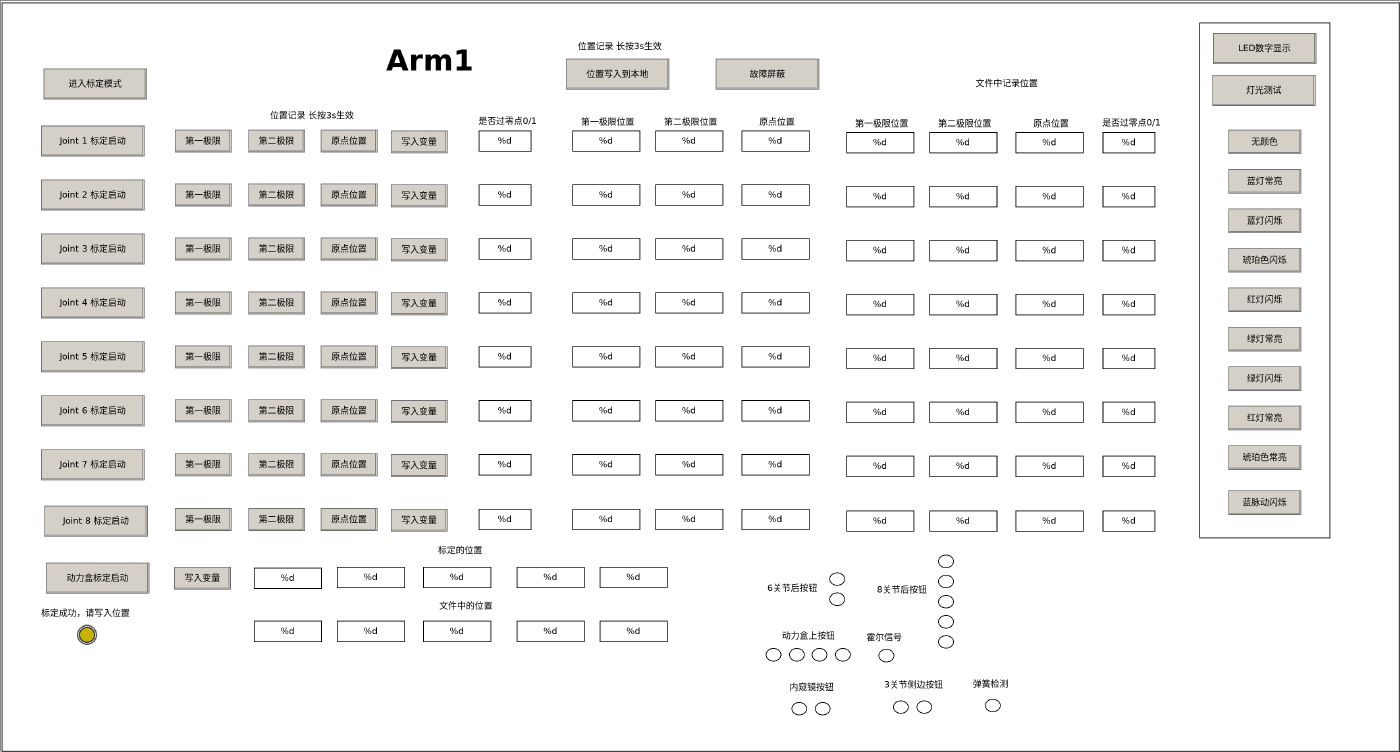
VISUALIZATION arm1Cail  // 1737x934
    Rectangle (2,3 1735x931)
    Button (54,85 128x38), "进入标定模式", colour toggle: GVL_armCali.g_armEnterCaliMode[1]
        toggle GVL_armCali.g_armEnterCaliMode[1]
    Button (51,156 128x38), "Joint 1 标定启动", colour toggle: GVL_armCali.g_jointIntoCaliState[1][1]
        toggle GVL_armCali.g_jointIntoCaliState[1][1]
    Label (435,49 197x52), "Arm1"
    Button (51,223 128x38), "Joint 2 标定启动", colour toggle: GVL_armCali.g_jointIntoCaliState[1][2]
        toggle GVL_armCali.g_jointIntoCaliState[1][2]
    Button (217,161 70x28), "第一极限", colour toggle: GVL_armCali.g_linkEncFristCaliTrigger[1][1]
        tap GVL_armCali.g_linkEncFristPosCali[1][1]
    Button (308,161 70x28), "第二极限", colour toggle: GVL_armCali.g_linkEncSecondCaliTrigger[1][1]
        tap GVL_armCali.g_linkEncSecondPosCali[1][1]
    Rectangle (594,162 65x26), "%d", text variable: GVL_armCali.g_linkZeroCrossOrNot[1][1]
    Label (589,139 82x23), "是否过零点0/1"
    Rectangle (710,162 84x26), "%d", text variable: GVL_armCali.g_linkLimitFristPos[1][1]
    Label (713,140 82x23), "第一极限位置"
    Rectangle (813,162 84x26), "%d", text variable: GVL_armCali.g_linkLimitSecondPos[1][1]
    Label (816,140 82x23), "第二极限位置"
    Label (312,132 150x23), "位置记录 长按3s生效"
    Rectangle (920,162 84x26), "%d", text variable: GVL_armCali.g_linkHomePos[1][1]
    Label (923,140 82x23), "原点位置"
    Button (398,161 70x28), "原点位置", colour toggle: GVL_armCali.g_linkEncHomePosCaliTrigger[1][1]
        tap GVL_armCali.g_linkEncHomePosCali[1][1]
    Button (702,73 128x38), "位置写入到本地", colour toggle: GVL_armCali.g_caliDataWriteTrigger[1]
        tap GVL_armCali.g_caliDataWrite[1]
    Label (694,46 150x23), "位置记录 长按3s生效"
    Button (217,228 70x28), "第一极限", colour toggle: GVL_armCali.g_linkEncFristCaliTrigger[1][2]
        tap GVL_armCali.g_linkEncFristPosCali[1][2]
    Button (308,228 70x28), "第二极限", colour toggle: GVL_armCali.g_linkEncSecondCaliTrigger[1][2]
        tap GVL_armCali.g_linkEncSecondPosCali[1][2]
    Rectangle (594,229 65x26), "%d", text variable: GVL_armCali.g_linkZeroCrossOrNot[1][2]
    Rectangle (710,229 84x26), "%d", text variable: GVL_armCali.g_linkLimitFristPos[1][2]
    Rectangle (813,229 84x26), "%d", text variable: GVL_armCali.g_linkLimitSecondPos[1][2]
    Rectangle (920,229 84x26), "%d", text variable: GVL_armCali.g_linkHomePos[1][2]
    Button (398,228 70x28), "原点位置", colour toggle: GVL_armCali.g_linkEncHomePosCaliTrigger[1][2]
        tap GVL_armCali.g_linkEncHomePosCali[1][2]
    Button (51,290 128x38), "Joint 3 标定启动", colour toggle: GVL_armCali.g_jointIntoCaliState[1][3]
        toggle GVL_armCali.g_jointIntoCaliState[1][3]
    Button (217,295 70x28), "第一极限", colour toggle: GVL_armCali.g_linkEncFristCaliTrigger[1][3]
        tap GVL_armCali.g_linkEncFristPosCali[1][3]
    Button (308,295 70x28), "第二极限", colour toggle: GVL_armCali.g_linkEncSecondCaliTrigger[1][3]
        tap GVL_armCali.g_linkEncSecondPosCali[1][3]
    Rectangle (594,296 65x26), "%d", text variable: GVL_armCali.g_linkZeroCrossOrNot[1][3]
    Rectangle (710,296 84x26), "%d", text variable: GVL_armCali.g_linkLimitFristPos[1][3]
    Rectangle (813,296 84x26), "%d", text variable: GVL_armCali.g_linkLimitSecondPos[1][3]
    Rectangle (920,296 84x26), "%d", text variable: GVL_armCali.g_linkHomePos[1][3]
    Button (398,295 70x28), "原点位置", colour toggle: GVL_armCali.g_linkEncHomePosCaliTrigger[1][3]
        tap GVL_armCali.g_linkEncHomePosCali[1][3]
    Button (51,357 128x38), "Joint 4 标定启动", colour toggle: GVL_armCali.g_jointIntoCaliState[1][4]
        toggle GVL_armCali.g_jointIntoCaliState[1][4]
    Button (217,362 70x28), "第一极限", colour toggle: GVL_armCali.g_linkEncFristCaliTrigger[1][4]
        tap GVL_armCali.g_linkEncFristPosCali[1][4]
    Button (308,362 70x28), "第二极限", colour toggle: GVL_armCali.g_linkEncSecondCaliTrigger[1][4]
        tap GVL_armCali.g_linkEncSecondPosCali[1][4]
    Rectangle (594,363 65x26), "%d", text variable: GVL_armCali.g_linkZeroCrossOrNot[1][4]
    Rectangle (710,363 84x26), "%d", text variable: GVL_armCali.g_linkLimitFristPos[1][4]
    Rectangle (813,363 84x26), "%d", text variable: GVL_armCali.g_linkLimitSecondPos[1][4]
    Rectangle (920,363 84x26), "%d", text variable: GVL_armCali.g_linkHomePos[1][4]
    Button (398,362 70x28), "原点位置", colour toggle: GVL_armCali.g_linkEncHomePosCaliTrigger[1][4]
        tap GVL_armCali.g_linkEncHomePosCali[1][4]
    Button (51,424 128x38), "Joint 5 标定启动", colour toggle: GVL_armCali.g_jointIntoCaliState[1][5]
        toggle GVL_armCali.g_jointIntoCaliState[1][5]
    Button (217,429 70x28), "第一极限", colour toggle: GVL_armCali.g_linkEncFristCaliTrigger[1][5]
        tap GVL_armCali.g_linkEncFristPosCali[1][5]
    Button (308,429 70x28), "第二极限", colour toggle: GVL_armCali.g_linkEncSecondCaliTrigger[1][5]
        tap GVL_armCali.g_linkEncSecondPosCali[1][5]
    Rectangle (594,430 65x26), "%d", text variable: GVL_armCali.g_linkZeroCrossOrNot[1][5]
    Rectangle (710,430 84x26), "%d", text variable: GVL_armCali.g_linkLimitFristPos[1][5]
    Rectangle (813,430 84x26), "%d", text variable: GVL_armCali.g_linkLimitSecondPos[1][5]
    Rectangle (920,430 84x26), "%d", text variable: GVL_armCali.g_linkHomePos[1][5]
    Button (398,429 70x28), "原点位置", colour toggle: GVL_armCali.g_linkEncHomePosCaliTrigger[1][5]
        tap GVL_armCali.g_linkEncHomePosCali[1][5]
    Button (51,491 128x38), "Joint 6 标定启动", colour toggle: GVL_armCali.g_jointIntoCaliState[1][6]
        toggle GVL_armCali.g_jointIntoCaliState[1][6]
    Button (217,496 70x28), "第一极限", colour toggle: GVL_armCali.g_linkEncFristCaliTrigger[1][6]
        tap GVL_armCali.g_linkEncFristPosCali[1][6]
    Button (308,496 70x28), "第二极限", colour toggle: GVL_armCali.g_linkEncSecondCaliTrigger[1][6]
        tap GVL_armCali.g_linkEncSecondPosCali[1][6]
    Rectangle (594,497 65x26), "%d", text variable: GVL_armCali.g_linkZeroCrossOrNot[1][6]
    Rectangle (710,497 84x26), "%d", text variable: GVL_armCali.g_linkLimitFristPos[1][6]
    Rectangle (813,497 84x26), "%d", text variable: GVL_armCali.g_linkLimitSecondPos[1][6]
    Rectangle (920,497 84x26), "%d", text variable: GVL_armCali.g_linkHomePos[1][6]
    Button (398,496 70x28), "原点位置", colour toggle: GVL_armCali.g_linkEncHomePosCaliTrigger[1][6]
        tap GVL_armCali.g_linkEncHomePosCali[1][6]
    Button (51,558 128x38), "Joint 7 标定启动", colour toggle: GVL_armCali.g_jointIntoCaliState[1][7]
        toggle GVL_armCali.g_jointIntoCaliState[1][7]
    Button (217,563 70x28), "第一极限", colour toggle: GVL_armCali.g_linkEncFristCaliTrigger[1][7]
        tap GVL_armCali.g_linkEncFristPosCali[1][7]
    Button (308,563 70x28), "第二极限", colour toggle: GVL_armCali.g_linkEncSecondCaliTrigger[1][7]
        tap GVL_armCali.g_linkEncSecondPosCali[1][7]
    Rectangle (594,564 65x26), "%d", text variable: GVL_armCali.g_linkZeroCrossOrNot[1][7]
    Rectangle (710,564 84x26), "%d", text variable: GVL_armCali.g_linkLimitFristPos[1][7]
    Rectangle (813,564 84x26), "%d", text variable: GVL_armCali.g_linkLimitSecondPos[1][7]
    Rectangle (920,564 84x26), "%d", text variable: GVL_armCali.g_linkHomePos[1][7]
    Button (398,563 70x28), "原点位置", colour toggle: GVL_armCali.g_linkEncHomePosCaliTrigger[1][7]
        tap GVL_armCali.g_linkEncHomePosCali[1][7]
    Button (55,628 128x38), "Joint 8 标定启动", colour toggle: GVL_armCali.g_jointIntoCaliState[1][8]
        toggle GVL_armCali.g_jointIntoCaliState[1][8]
    Button (217,631 70x28), "第一极限", colour toggle: GVL_armCali.g_linkEncFristCaliTrigger[1][8]
        tap GVL_armCali.g_linkEncFristPosCali[1][8]
    Button (308,631 70x28), "第二极限", colour toggle: GVL_armCali.g_linkEncSecondCaliTrigger[1][8]
        tap GVL_armCali.g_linkEncSecondPosCali[1][8]
    Rectangle (594,632 65x26), "%d", text variable: GVL_armCali.g_linkZeroCrossOrNot[1][8]
    Rectangle (710,632 84x26), "%d", text variable: GVL_armCali.g_linkLimitFristPos[1][8]
    Rectangle (813,632 84x26), "%d", text variable: GVL_armCali.g_linkLimitSecondPos[1][8]
    Rectangle (920,632 84x26), "%d", text variable: GVL_armCali.g_linkHomePos[1][8]
    Button (398,631 70x28), "原点位置", colour toggle: GVL_armCali.g_linkEncHomePosCaliTrigger[1][8]
        tap GVL_armCali.g_linkEncHomePosCali[1][8]
    Rectangle (1050,164 84x26), "%d", text variable: GVL_SetupJointEncoderCaliData.g_minLinkEncoder[1,1]
    Label (1053,142 82x23), "第一极限位置"
    Rectangle (1153,164 84x26), "%d", text variable: GVL_SetupJointEncoderCaliData.g_maxLinkEncoder[1,1]
    Label (1156,142 82x23), "第二极限位置"
    Rectangle (1260,164 84x26), "%d", text variable: GVL_SetupJointEncoderCaliData.g_caliLinkEncoder[1,1]
    Label (1263,142 82x23), "原点位置"
    Rectangle (1050,231 84x26), "%d", text variable: GVL_SetupJointEncoderCaliData.g_minLinkEncoder[1,2]
    Rectangle (1153,231 84x26), "%d", text variable: GVL_SetupJointEncoderCaliData.g_maxLinkEncoder[1,2]
    Rectangle (1260,231 84x26), "%d", text variable: GVL_SetupJointEncoderCaliData.g_caliLinkEncoder[1,2]
    Rectangle (1050,298 84x26), "%d", text variable: GVL_SetupJointEncoderCaliData.g_minLinkEncoder[1,3]
    Rectangle (1153,298 84x26), "%d", text variable: GVL_SetupJointEncoderCaliData.g_maxLinkEncoder[1,3]
    Rectangle (1260,298 84x26), "%d", text variable: GVL_SetupJointEncoderCaliData.g_caliLinkEncoder[1,3]
    Rectangle (1050,365 84x26), "%d", text variable: GVL_SetupJointEncoderCaliData.g_minLinkEncoder[1,4]
    Rectangle (1153,365 84x26), "%d", text variable: GVL_SetupJointEncoderCaliData.g_maxLinkEncoder[1,4]
    Rectangle (1260,365 84x26), "%d", text variable: GVL_SetupJointEncoderCaliData.g_caliLinkEncoder[1,4]
    Rectangle (1050,432 84x26), "%d", text variable: GVL_SetupJointEncoderCaliData.g_minLinkEncoder[1,5]
    Rectangle (1153,432 84x26), "%d", text variable: GVL_SetupJointEncoderCaliData.g_maxLinkEncoder[1,5]
    Rectangle (1260,432 84x26), "%d", text variable: GVL_SetupJointEncoderCaliData.g_caliLinkEncoder[1,5]
    Rectangle (1050,499 84x26), "%d", text variable: GVL_SlaveJointEncoderCaliData.g_minLinkEncoder[1,1]
    Rectangle (1153,499 84x26), "%d", text variable: GVL_SlaveJointEncoderCaliData.g_maxLinkEncoder[1,1]
    Rectangle (1260,499 84x26), "%d", text variable: GVL_SlaveJointEncoderCaliData.g_caliLinkEncoder[1,1]
    Rectangle (1050,566 84x26), "%d", text variable: GVL_SlaveJointEncoderCaliData.g_minLinkEncoder[1,2]
    Rectangle (1153,566 84x26), "%d", text variable: GVL_SlaveJointEncoderCaliData.g_maxLinkEncoder[1,2]
    Rectangle (1260,566 84x26), "%d", text variable: GVL_SlaveJointEncoderCaliData.g_caliLinkEncoder[1,2]
    Rectangle (1050,634 84x26), "%d", text variable: GVL_SlaveJointEncoderCaliData.g_minLinkEncoder[1,3]
    Rectangle (1153,634 84x26), "%d", text variable: GVL_SlaveJointEncoderCaliData.g_maxLinkEncoder[1,3]
    Rectangle (1260,634 84x26), "%d", text variable: GVL_SlaveJointEncoderCaliData.g_caliLinkEncoder[1,3]
    Label (1174,92 150x23), "文件中记录位置"
    Rectangle (1368,164 65x26), "%d", text variable: GVL_SetupJointEncoderCaliData.g_linkEncZeroCross[1,1]
    Label (1363,141 82x23), "是否过零点0/1"
    Rectangle (1368,231 65x26), "%d", text variable: GVL_SetupJointEncoderCaliData.g_linkEncZeroCross[1,2]
    Rectangle (1368,298 65x26), "%d", text variable: GVL_SetupJointEncoderCaliData.g_linkEncZeroCross[1,3]
    Rectangle (1368,365 65x26), "%d", text variable: GVL_SetupJointEncoderCaliData.g_linkEncZeroCross[1,4]
    Rectangle (1368,432 65x26), "%d", text variable: GVL_SetupJointEncoderCaliData.g_linkEncZeroCross[1,5]
    Rectangle (1368,499 65x26), "%d", text variable: GVL_SlaveJointEncoderCaliData.g_linkEncZeroCross[1,1]
    Rectangle (1368,566 65x26), "%d", text variable: GVL_SlaveJointEncoderCaliData.g_linkEncZeroCross[1,2]
    Rectangle (1368,634 65x26), "%d", text variable: GVL_SlaveJointEncoderCaliData.g_linkEncZeroCross[1,3]
    Button (485,162 70x28), "写入变量", colour toggle: GVL_armCali.g_linkPosWriteCaliDataTrigger[1][1]
        tap GVL_armCali.g_linkPosWriteCaliData[1][1]
    Button (485,229 70x28), "写入变量", colour toggle: GVL_armCali.g_linkPosWriteCaliDataTrigger[1][2]
        tap GVL_armCali.g_linkPosWriteCaliData[1][2]
    Button (485,296 70x28), "写入变量", colour toggle: GVL_armCali.g_linkPosWriteCaliDataTrigger[1][3]
        tap GVL_armCali.g_linkPosWriteCaliData[1][3]
    Button (485,363 70x28), "写入变量", colour toggle: GVL_armCali.g_linkPosWriteCaliDataTrigger[1][4]
        tap GVL_armCali.g_linkPosWriteCaliData[1][4]
    Button (485,430 70x28), "写入变量", colour toggle: GVL_armCali.g_linkPosWriteCaliDataTrigger[1][5]
        tap GVL_armCali.g_linkPosWriteCaliData[1][5]
    Button (485,497 70x28), "写入变量", colour toggle: GVL_armCali.g_linkPosWriteCaliDataTrigger[1][6]
        tap GVL_armCali.g_linkPosWriteCaliData[1][6]
    Button (485,564 70x28), "写入变量", colour toggle: GVL_armCali.g_linkPosWriteCaliDataTrigger[1][7]
        tap GVL_armCali.g_linkPosWriteCaliData[1][7]
    Button (485,632 70x28), "写入变量", colour toggle: GVL_armCali.g_linkPosWriteCaliDataTrigger[1][8]
        tap GVL_armCali.g_linkPosWriteCaliData[1][8]
    Button (57,699 128x38), "动力盒标定启动", colour toggle: GVL_armCali.g_powerBoxCali[1]
        toggle GVL_armCali.g_powerBoxCali[1]
    Lamp1 (88,774 40x29), invisible if: GVL_armCali.g_powerBoxCalicomplete[1], style: Lamp-Lamp1-Yellow
    Label (31,750 150x23), "标定成功，请写入位置"
    Button (216,704 70x28), "写入变量", colour toggle: GVL_armCali.g_powerBoxPosWriteTrigger[1]
        tap GVL_armCali.g_powerBoxPosWrite[1]
    Rectangle (315,705 84x26), "%d", text variable: GVL_armCali.g_powerBoxLinkHomePos[1][1]
    Rectangle (418,704 84x26), "%d", text variable: GVL_armCali.g_powerBoxLinkHomePos[1][2]
    Rectangle (525,704 84x26), "%d", text variable: GVL_armCali.g_powerBoxLinkHomePos[1][3]
    Rectangle (641,704 84x26), "%d", text variable: GVL_armCali.g_powerBoxLinkHomePos[1][4]
    Rectangle (744,704 84x26), "%d", text variable: GVL_armCali.g_powerBoxLinkHomePos[1][5]
    Rectangle (315,771 84x26), "%d", text variable: GVL_SlaveJointEncoderCaliData.g_caliLinkEncoder[1,4]
    Rectangle (418,771 84x26), "%d", text variable: GVL_SlaveJointEncoderCaliData.g_caliLinkEncoder[1,5]
    Rectangle (525,771 84x26), "%d", text variable: GVL_SlaveJointEncoderCaliData.g_caliLinkEncoder[1,6]
    Rectangle (641,771 84x26), "%d", text variable: GVL_SlaveJointEncoderCaliData.g_caliLinkEncoder[1,7]
    Rectangle (744,771 84x26), "%d", text variable: GVL_SlaveJointEncoderCaliData.g_caliLinkEncoder[1,8]
    Label (503,741 150x23), "文件中的位置"
    Label (496,672 150x23), "标定的位置"
    Label (943,719 80x23), "6关节后按钮"
    Ellipse (1029,736 19x16), colour toggle: GVL_IO.g_joint6IO[1][2]
    Ellipse (1029,711 19x16), colour toggle: GVL_IO.g_joint6IO[1][1]
    Label (1079,721 80x23), "8关节后按钮"
    Ellipse (1164,714 19x16), colour toggle: GVL_IO.g_joint8IO[1][2]
    Ellipse (1164,689 19x16), colour toggle: GVL_IO.g_joint8IO[1][1]
    Ellipse (1164,764 19x16), colour toggle: GVL_IO.g_joint8IO[1][4]
    Ellipse (1164,739 19x16), colour toggle: GVL_IO.g_joint8IO[1][3]
    Label (963,778 80x23), "动力盒上按钮"
    Ellipse (950,805 19x16), colour toggle: GVL_IO.g_jointPowerBoxIO[1][1]
    Ellipse (979,805 19x16), colour toggle: GVL_IO.g_jointPowerBoxIO[1][2]
    Ellipse (1007,805 19x16), colour toggle: GVL_IO.g_jointPowerBoxIO[1][3]
    Ellipse (1036,805 19x16), colour toggle: GVL_IO.g_jointPowerBoxIO[1][4]
    Label (967,842 80x23), "内窥镜按钮"
    Ellipse (982,872 19x16), colour toggle: GVL_IO.g_endoscopeSingle[1][1]
    Ellipse (1011,872 19x16), colour toggle: GVL_IO.g_endoscopeSingle[1][2]
    Ellipse (1164,789 19x16), colour toggle: GVL_IO.g_joint8IO[1][5]
    Ellipse (1090,806 19x16), colour toggle: GVL_IO.g_jointPowerBoxIO[1][5]
    Label (1057,780 80x23), "霍尔信号"
    Rectangle (1488,28 162x640)
    Button (1524,161 90x30), "无颜色", colour toggle: GVL_IO.g_armLight_PowerOff[1]
        toggle GVL_IO.g_armLight_PowerOff[1]
    Button (1524,210 90x30), "蓝灯常亮", colour toggle: GVL_IO.g_armLight_BlueOn[1]
        toggle GVL_IO.g_armLight_BlueOn[1]
    Button (1524,259 90x30), "蓝灯闪烁", colour toggle: GVL_IO.g_armLight_BlueBlink[1]
        toggle GVL_IO.g_armLight_BlueBlink[1]
    Button (1524,308 90x30), "琥珀色闪烁", colour toggle: GVL_IO.g_armLight_AmberBlink[1]
        toggle GVL_IO.g_armLight_AmberBlink[1]
    Button (1524,357 90x30), "红灯闪烁", colour toggle: GVL_IO.g_armLight_RedBlink[1]
        toggle GVL_IO.g_armLight_RedBlink[1]
    Button (1524,406 90x30), "绿灯常亮", colour toggle: GVL_IO.g_armLight_GreenOn[1]
        toggle GVL_IO.g_armLight_GreenOn[1]
    Button (1524,455 90x30), "绿灯闪烁", colour toggle: GVL_IO.g_armLight_GreenBlink[1]
        toggle GVL_IO.g_armLight_GreenBlink[1]
    Button (1504,93 128x38), "灯光测试", colour toggle: GVL_IO.g_lightTest[1]
        toggle GVL_IO.g_lightTest[1]
    Button (1524,504 90x30), "红灯常亮", colour toggle: GVL_IO.g_armLight_redOn[1]
        toggle GVL_IO.g_armLight_redOn[1]
    Button (1524,553 90x30), "琥珀色常亮", colour toggle: GVL_IO.g_armLight_AmberOn[1]
        toggle GVL_IO.g_armLight_AmberOn[1]
    Button (1524,609 90x30), "蓝脉动闪烁", colour toggle: GVL_IO.g_armLight_BluePulse[1]
        toggle GVL_IO.g_armLight_BluePulse[1]
    Button (1505,41 128x38), "LED数字显示", colour toggle: GVL_IO.g_LEDValueDisplay[1]
        toggle GVL_IO.g_LEDValueDisplay[1]
    Label (1076,839 115x23), "3关节侧边按钮"
    Ellipse (1108,870 19x16), colour toggle: GVL_IO.g_asepticMegnetCheck[1][1]
    Ellipse (1137,870 19x16), colour toggle: GVL_IO.g_asepticMegnetCheck[1][2]
    Ellipse (1222,868 19x16)
    Label (1189,838 80x23), "弹簧检测"
    Button (888,73 128x38), "故障屏蔽", colour toggle: g_specialSignal.m_faultMask[1]
        toggle g_specialSignal.m_faultMask[1]
END_VISUALIZATION

(* stored: Version 1.1.0.1, ProductVersion 3.1.4024.11
   Visu arm1Cail: Id {b447a79d-70e3-4b30-9c37-cd0deb6bd1d5} *)
